// Mitsubishi GX Works2 project: connection   PLC: Q03UDV

PROGRAM MAIN
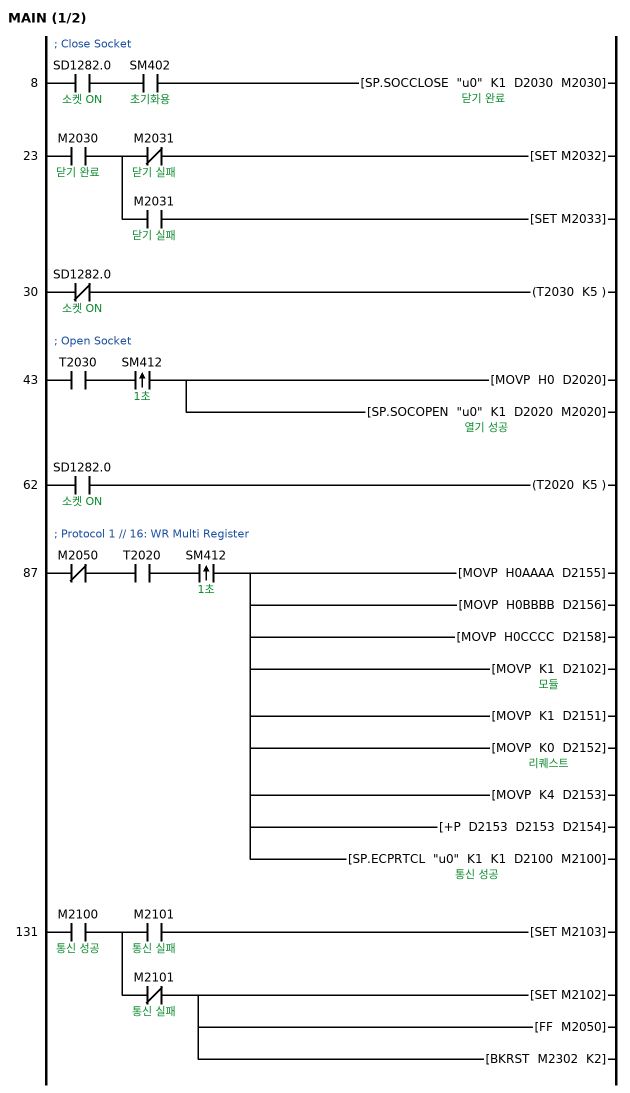
; Close Socket
8     LD      SD1282.0  ; 소켓 ON
      AND     SM402  ; 초기화용
      SP.SOCCLOSE "u0" K1 D2030 M2030  ; 닫기 완료
23    LD      M2030  ; 닫기 완료
      MPS
      ANI     M2031  ; 닫기 실패
      SET     M2032
      MPP
      AND     M2031  ; 닫기 실패
      SET     M2033
30    LDI     SD1282.0  ; 소켓 ON
      OUT     T2030 K5
; Open Socket
43    LD      T2030
      ANDP    SM412  ; 1초
      MOVP    H0 D2020
      SP.SOCOPEN "u0" K1 D2020 M2020  ; 열기 성공
62    LD      SD1282.0  ; 소켓 ON
      OUT     T2020 K5
; Protocol 1 // 16: WR Multi Register
87    LDI     M2050
      AND     T2020
      ANDP    SM412  ; 1초
      MOVP    H0AAAA D2155
      MOVP    H0BBBB D2156
      MOVP    H0CCCC D2158
      MOVP    K1 D2102  ; 모듈
      MOVP    K1 D2151
      MOVP    K0 D2152  ; 리퀘스트
      MOVP    K4 D2153
      +P      D2153 D2153 D2154
      SP.ECPRTCL "u0" K1 K1 D2100 M2100  ; 통신 성공
131   LD      M2100  ; 통신 성공
      MPS
      AND     M2101  ; 통신 실패
      SET     M2103
      MPP
      ANI     M2101  ; 통신 실패
      SET     M2102
      FF      M2050
      BKRST   M2302 K2
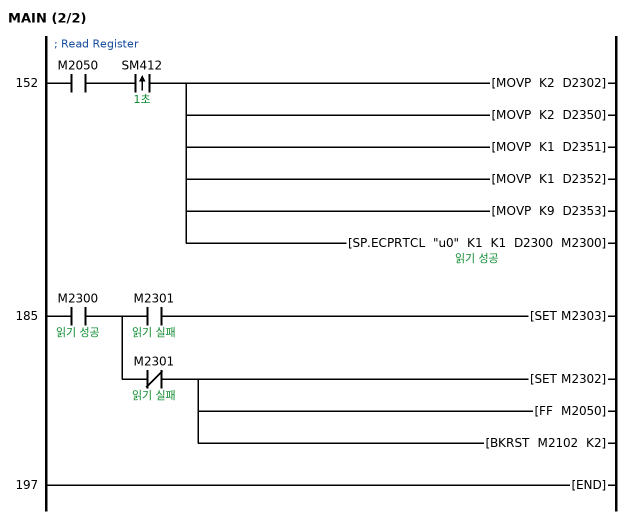
; Read Register
152   LD      M2050
      ANDP    SM412  ; 1초
      MOVP    K2 D2302
      MOVP    K2 D2350
      MOVP    K1 D2351
      MOVP    K1 D2352
      MOVP    K9 D2353
      SP.ECPRTCL "u0" K1 K1 D2300 M2300  ; 읽기 성공
185   LD      M2300  ; 읽기 성공
      MPS
      AND     M2301  ; 읽기 실패
      SET     M2303
      MPP
      ANI     M2301  ; 읽기 실패
      SET     M2302
      FF      M2050
      BKRST   M2102 K2
197   END
END_PROGRAM

// device comments not shown above
D2101  ; 트랜잭션
